// TIA Portal V18 export
// export: Created 2025-12-01T17:51:11.0018068Z, ExportSetting None, DisplayName Totally Integrated Automation Portal, DisplayVersion V18 Update 5, DisplayName TIA Portal Openness, DisplayVersion V18 Update 5, DisplayName TIA Portal Teamcenter Gateway, DisplayVersion V18, DisplayName TIA Portal Version Control Interface, DisplayVersion V18, DisplayName STEP 7 Professional, DisplayVersion V18 Update 5, DisplayName STEP 7 Safety, DisplayVersion V18, DisplayName WinCC Professional, DisplayVersion V18 Update 5
DATA_BLOCK "HMISystemDB"   // DB2201
{ S7_Optimized_Access := 'FALSE' }
// stored: AutoNumber false
   VAR RETAIN
      DisplayRows : Int;
      MaxPage : Int;
      Rows : Int;
      UnEnableGroup : Bool;
      DisplaySymbol : Bool;
      "DisplaySymbol Time" : Int;
      SymbolText : Array[1..4] of Int;
      HMICylinderBypass : Array[1..50] of Struct
         "BY" : Array[1..50] of Int;
      END_STRUCT;
      HMI_Axis : "HMI_Axis";
   END_VAR
BEGIN
   HMI_Axis.INPUT.Axis_ID := 1;
END_DATA_BLOCK
